{attribute 'pack_mode' := '1'}
TYPE  ST_HexColor:
STRUCT
	
	(*	Color Hexcode...[generiert aus .net]		*)
	ActiveBorder :DINT:=16#D4D0C8;
	ActiveCaption :DINT:=16#0054E3;
	ActiveCaptionText :DINT:=16#FFFFFF;
	AliceBlue :DINT:=16#F0F8FF;
	AntiqueWhite :DINT:=16#FAEBD7;
	AppWorkspace :DINT:=16#808080;
	Aqua :DINT:=16#00FFFF;
	Aquamarine :DINT:=16#7FFFD4;
	Azure :DINT:=16#F0FFFF;
	Beige :DINT:=16#F5F5DC;
	Bisque :DINT:=16#FFE4C4;
	Black :DINT:=16#000000;
	BlanchedAlmond :DINT:=16#FFEBCD;
	Blue :DINT:=16#0000FF;
	BlueViolet :DINT:=16#8A2BE2;
	Brown :DINT:=16#A52A2A;
	BurlyWood :DINT:=16#DEB887;
	ButtonFace :DINT:=16#ECE9D8;
	ButtonHighlight :DINT:=16#FFFFFF;
	ButtonShadow :DINT:=16#ACA899;
	CadetBlue :DINT:=16#5F9EA0;
	Chartreuse :DINT:=16#7FFF00;
	Chocolate :DINT:=16#D2691E;
	Control :DINT:=16#ECE9D8;
	ControlDark :DINT:=16#ACA899;
	ControlDarkDark :DINT:=16#716F64;
	ControlLight :DINT:=16#F1EFE2;
	ControlLightLight :DINT:=16#FFFFFF;
	ControlText :DINT:=16#000000;
	Coral :DINT:=16#FF7F50;
	CornflowerBlue :DINT:=16#6495ED;
	Cornsilk :DINT:=16#FFF8DC;
	Crimson :DINT:=16#DC143C;
	Cyan :DINT:=16#00FFFF;
	DarkBlue :DINT:=16#00008B;
	DarkCyan :DINT:=16#008B8B;
	DarkGoldenrod :DINT:=16#B8860B;
	DarkGray :DINT:=16#A9A9A9;
	DarkGreen :DINT:=16#006400;
	DarkKhaki :DINT:=16#BDB76B;
	DarkMagenta :DINT:=16#8B008B;
	DarkOliveGreen :DINT:=16#556B2F;
	DarkOrange :DINT:=16#FF8C00;
	DarkOrchid :DINT:=16#9932CC;
	DarkRed :DINT:=16#8B0000;
	DarkSalmon :DINT:=16#E9967A;
	DarkSeaGreen :DINT:=16#8FBC8B;
	DarkSlateBlue :DINT:=16#483D8B;
	DarkSlateGray :DINT:=16#2F4F4F;
	DarkTurquoise :DINT:=16#00CED1;
	DarkViolet :DINT:=16#9400D3;
	DeepPink :DINT:=16#FF1493;
	DeepSkyBlue :DINT:=16#00BFFF;
	Desktop :DINT:=16#004E98;
	DimGray :DINT:=16#696969;
	DodgerBlue :DINT:=16#1E90FF;
	Firebrick :DINT:=16#B22222;
	FloralWhite :DINT:=16#FFFAF0;
	ForestGreen :DINT:=16#228B22;
	Fuchsia :DINT:=16#FF00FF;
	Gainsboro :DINT:=16#DCDCDC;
	GhostWhite :DINT:=16#F8F8FF;
	Gold :DINT:=16#FFD700;
	Goldenrod :DINT:=16#DAA520;
	GradientActiveCaption :DINT:=16#3D95FF;
	GradientInactiveCaption :DINT:=16#9DB9EB;
	Gray :DINT:=16#808080;
	GrayText :DINT:=16#ACA899;
	Green :DINT:=16#008000;
	GreenYellow :DINT:=16#ADFF2F;
	Highlight :DINT:=16#316AC5;
	HighlightText :DINT:=16#FFFFFF;
	Honeydew :DINT:=16#F0FFF0;
	HotPink :DINT:=16#FF69B4;
	HotTrack :DINT:=16#000080;
	InactiveBorder :DINT:=16#D4D0C8;
	InactiveCaption :DINT:=16#7A96DF;
	InactiveCaptionText :DINT:=16#D8E4F8;
	IndianRed :DINT:=16#CD5C5C;
	Indigo :DINT:=16#4B0082;
	Info :DINT:=16#FFFFE1;
	InfoText :DINT:=16#000000;
	Ivory :DINT:=16#FFFFF0;
	Khaki :DINT:=16#F0E68C;
	Lavender :DINT:=16#E6E6FA;
	LavenderBlush :DINT:=16#FFF0F5;
	LawnGreen :DINT:=16#7CFC00;
	LemonChiffon :DINT:=16#FFFACD;
	LightBlue :DINT:=16#ADD8E6;
	LightCoral :DINT:=16#F08080;
	LightCyan :DINT:=16#E0FFFF;
	LightGoldenrodYellow :DINT:=16#FAFAD2;
	LightGray :DINT:=16#D3D3D3;
	LightGreen :DINT:=16#90EE90;
	LightPink :DINT:=16#FFB6C1;
	LightSalmon :DINT:=16#FFA07A;
	LightSeaGreen :DINT:=16#20B2AA;
	LightSkyBlue :DINT:=16#87CEFA;
	LightSlateGray :DINT:=16#778899;
	LightSteelBlue :DINT:=16#B0C4DE;
	LightYellow :DINT:=16#FFFFE0;
	Lime :DINT:=16#00FF00;
	LimeGreen :DINT:=16#32CD32;
	Linen :DINT:=16#FAF0E6;
	Magenta :DINT:=16#FF00FF;
	Maroon :DINT:=16#800000;
	MediumAquamarine :DINT:=16#66CDAA;
	MediumBlue :DINT:=16#0000CD;
	MediumOrchid :DINT:=16#BA55D3;
	MediumPurple :DINT:=16#9370DB;
	MediumSeaGreen :DINT:=16#3CB371;
	MediumSlateBlue :DINT:=16#7B68EE;
	MediumSpringGreen :DINT:=16#00FA9A;
	MediumTurquoise :DINT:=16#48D1CC;
	MediumVioletRed :DINT:=16#C71585;
	Menu :DINT:=16#FFFFFF;
	MenuBar :DINT:=16#ECE9D8;
	MenuHighlight :DINT:=16#316AC5;
	MenuText :DINT:=16#000000;
	MidnightBlue :DINT:=16#191970;
	MintCream :DINT:=16#F5FFFA;
	MistyRose :DINT:=16#FFE4E1;
	Moccasin :DINT:=16#FFE4B5;
	NavajoWhite :DINT:=16#FFDEAD;
	Navy :DINT:=16#000080;
	OldLace :DINT:=16#FDF5E6;
	Olive :DINT:=16#808000;
	OliveDrab :DINT:=16#6B8E23;
	Orange :DINT:=16#FFA500;
	OrangeRed :DINT:=16#FF4500;
	Orchid :DINT:=16#DA70D6;
	PaleGoldenrod :DINT:=16#EEE8AA;
	PaleGreen :DINT:=16#98FB98;
	PaleTurquoise :DINT:=16#AFEEEE;
	PaleVioletRed :DINT:=16#DB7093;
	PapayaWhip :DINT:=16#FFEFD5;
	PeachPuff :DINT:=16#FFDAB9;
	Peru :DINT:=16#CD853F;
	Pink :DINT:=16#FFC0CB;
	Plum :DINT:=16#DDA0DD;
	PowderBlue :DINT:=16#B0E0E6;
	Purple :DINT:=16#800080;
	Red :DINT:=16#FF0000;
	RosyBrown :DINT:=16#BC8F8F;
	RoyalBlue :DINT:=16#4169E1;
	SaddleBrown :DINT:=16#8B4513;
	Salmon :DINT:=16#FA8072;
	SandyBrown :DINT:=16#F4A460;
	ScrollBar :DINT:=16#D4D0C8;
	SeaGreen :DINT:=16#2E8B57;
	SeaShell :DINT:=16#FFF5EE;
	Sienna :DINT:=16#A0522D;
	Silver :DINT:=16#C0C0C0;
	SkyBlue :DINT:=16#87CEEB;
	SlateBlue :DINT:=16#6A5ACD;
	SlateGray :DINT:=16#708090;
	Snow :DINT:=16#FFFAFA;
	SpringGreen :DINT:=16#00FF7F;
	SteelBlue :DINT:=16#4682B4;
	TTAN :DINT:=16#D2B48C;
	Teal :DINT:=16#008080;
	Thistle :DINT:=16#D8BFD8;
	Tomato :DINT:=16#FF6347;
	//Transparent :DINT:=16#FFFFFF;
	Turquoise :DINT:=16#40E0D0;
	Violet :DINT:=16#EE82EE;
	Wheat :DINT:=16#F5DEB3;
	White :DINT:=16#FFFFFF;
	WhiteSmoke :DINT:=16#F5F5F5;
	Window :DINT:=16#FFFFFF;
	WindowFrame :DINT:=16#000000;
	WindowText :DINT:=16#000000;
	Yellow :DINT:=16#FFFF00;
	YellowGreen :DINT:=16#9ACD32;
	GrassGreen	: DINT := 16#ADE204;
END_STRUCT
END_TYPE

(* stored: Version 1.1.0.1, ProductVersion 3.1.4024.12
   DUT ST_HexColor: Id {f51d0fc1-b4bc-4cca-b33b-ce4417734537} *)
